// TIA Portal V21 export
VAR_GLOBAL   // PLC tag table "K_SegnaliMacchina"
END_VAR
VAR_GLOBAL CONSTANT   // user constants
   K_SegnaliMacchina_QCI : Int := 1;
   K_SegnaliMacchina_CFT : Int := 2;
END_VAR
